// SIMATIC S7-200 project (STEP 7-Micro/WIN), CPU 221 REL 01.10

ORGANIZATION_BLOCK MAIN:OB1
TITLE=PROGRAM COMMENTS
BEGIN
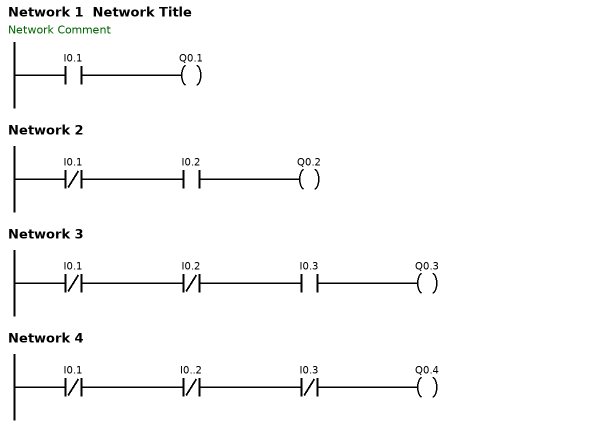
Network 1 // Network Title
// Network Comment
LD     I0.1
=      Q0.1
Network 2
LDN    I0.1
A      I0.2
=      Q0.2
Network 3
LDN    I0.1
AN     I0.2
A      I0.3
=      Q0.3
Network 4
// (network saved uncompiled; LAD cells follow)
// row 0: c0 -|/|- I0.1  c1 -|/|- I0..2  c2 -|/|- I0.3  c3 -( ) Q0.4
END_ORGANIZATION_BLOCK
